Yaskawa INFORM job: Program.JBI

/JOB
//NAME Program
//POS
///NPOS 3,0,0,0,0,0
///TOOL 9
///POSTYPE PULSE
///PULSE
C00000=-46,-7,-21,71,50,-303
///TOOL 9
///POSTYPE BASE
///RECTAN
///RCONF 0,0,0,0,0,0,0,0
C00001=200.000,250.000,348.735,-150.00,-0.00,180.00
C00002=200.000,200.000,262.132,-150.00,-0.00,180.00
//INST
///DATE 2022/10/28 12:16
///COMM Generated using RoboDK
///ATTR SC,RW,RJ
///GROUP1 RB1
NOP
'Program generated by RoboDK
MOVJ C00000 VJ=50.00
MOVL C00001 V=100.0
MOVL C00002 V=100.0
END
